// Mitsubishi GX Works2 project: PLC_status_fetcher   PLC: FX3G

PROGRAM MAIN
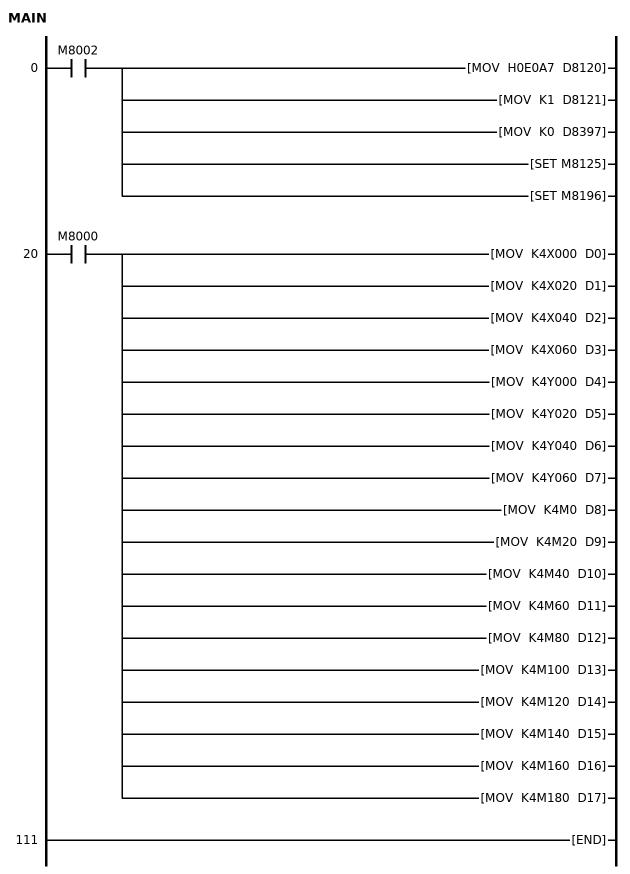
0     LD      M8002
      MOV     H0E0A7 D8120
      MOV     K1 D8121
      MOV     K0 D8397
      SET     M8125
      SET     M8196
20    LD      M8000
      MOV     K4X000 D0
      MOV     K4X020 D1
      MOV     K4X040 D2
      MOV     K4X060 D3
      MOV     K4Y000 D4
      MOV     K4Y020 D5
      MOV     K4Y040 D6
      MOV     K4Y060 D7
      MOV     K4M0 D8
      MOV     K4M20 D9
      MOV     K4M40 D10
      MOV     K4M60 D11
      MOV     K4M80 D12
      MOV     K4M100 D13
      MOV     K4M120 D14
      MOV     K4M140 D15
      MOV     K4M160 D16
      MOV     K4M180 D17
111   END
END_PROGRAM
